(* Logix 5000 project; controller ToyPlant Emulate 5570 rev 30.12; software revision 30.00 *)

TASK MainTask (continuous, watchdog 500 ms) : MainProgram

MODULES
   Local : Emulate 5570 (ICP 2, rev 30.12)
END_MODULES

PROGRAM MainProgram   (* main routine MainRoutine *)
VAR
   Action_000 : SFC_ACTION := (Count := 2);
   Action_001 : SFC_ACTION := (Count := 1);
   Action_002 : SFC_ACTION := (Count := 1);
   Action_003 : SFC_ACTION := (Count := 1);
   Action_004 : SFC_ACTION := (Count := 1);
   Action_005 : SFC_ACTION := (Count := 14);
   Action_006 : SFC_ACTION := (Count := 1);
   Action_007 : SFC_ACTION := (Count := 1);
   Action_008 : SFC_ACTION := (Count := 1);
   Action_009 : SFC_ACTION := (Count := 1);
   Action_010 : SFC_ACTION := (Count := 1);
   Action_011 : SFC_ACTION := (Count := 2);
   Action_012 : SFC_ACTION := (Count := 2);
   Action_013 : SFC_ACTION := (Count := 1);
   Action_014 : SFC_ACTION := (Count := 1);
   Action_015 : SFC_ACTION := (Count := 1);
   Action_016 : SFC_ACTION := (Count := 1);
   Action_017 : SFC_ACTION := (Count := 1);
   Action_018 : SFC_ACTION := (Count := 1);
   Action_019 : SFC_ACTION := (Count := 1);
   Action_020 : SFC_ACTION := (Count := 1);
   Action_021 : SFC_ACTION := (Status := 16#0020_0000, PauseTimer := 1, Count := 1);
   Action_022 : SFC_ACTION;
   Action_023 : SFC_ACTION;
   Action_024 : SFC_ACTION;
   Action_025 : SFC_ACTION;
   Action_026 : SFC_ACTION;
   Action_027 : SFC_ACTION;
   Action_028 : SFC_ACTION;
   Action_029 : SFC_ACTION := (Status := 16#0020_0000, PauseTimer := 1);
   Action_030 : SFC_ACTION := (Status := 16#0020_0000, PauseTimer := 1);
   Action_031 : SFC_ACTION := (Status := 16#0020_0000, PauseTimer := 1);
   Action_032 : SFC_ACTION := (Status := 16#0020_0000, PauseTimer := 1);
   Action_033 : SFC_ACTION := (Status := 16#0020_0000, PauseTimer := 1);
   Action_034 : SFC_ACTION := (Status := 16#0020_0000, PauseTimer := 1);
   Action_035 : SFC_ACTION := (Status := 16#0020_0000, PauseTimer := 1);
   Action_036 : SFC_ACTION := (Status := 16#0020_0000, PauseTimer := 1);
   Action_037 : SFC_ACTION := (Status := 16#0020_0000, PauseTimer := 1);
   Action_038 : SFC_ACTION := (Status := 16#0020_0000, PauseTimer := 1);
   Action_039 : SFC_ACTION := (Status := 16#0020_0000, PauseTimer := 1);
   Action_040 : SFC_ACTION := (Status := 16#0020_0000, PauseTimer := 1);
   Action_041 : SFC_ACTION := (Status := 16#0020_0000, PauseTimer := 1);
   Action_042 : SFC_ACTION := (Status := 16#0020_0000, PauseTimer := 1);
   Action_043 : SFC_ACTION := (Status := 16#0020_0000, PauseTimer := 1);
   Action_044 : SFC_ACTION := (Status := 16#0020_0000, PauseTimer := 1);
   Action_045 : SFC_ACTION := (Status := 16#0020_0000, PauseTimer := 1);
   BarcoReady : BOOL;
   CasaReady : BOOL;
   ContadorBarco : COUNTER := (PRE := 25);
   ContadorCasa : COUNTER := (PRE := 25);
   ContadorJuguetes : COUNTER := (PRE := 4);
   ContadorMoldes : COUNTER := (PRE := 4);
   ContadorMoto : COUNTER := (PRE := 25);
   MotoReady : BOOL;
   Off_ServoWorking : BOOL;
   PresetBarco : DINT := 1000;
   PresetCasa : DINT := 1000;
   PresetMoto : DINT := 1000;
   Step_000 : SFC_STEP := (T := 14169, TMax := 14169, Count := 2);
   Step_001 : SFC_STEP := (T := 1304, TMax := 1304, Count := 1);
   Step_002 : SFC_STEP := (T := 2486, TMax := 2486, Count := 1);
   Step_003 : SFC_STEP := (T := 21, TMax := 21, Count := 1);
   Step_004 : SFC_STEP := (T := 1039, TMax := 1039, Count := 1);
   Step_005 : SFC_STEP := (T := 21, TMax := 22, Count := 14);
   Step_006 : SFC_STEP := (T := 1975, TMax := 1975, Count := 1);
   Step_007 : SFC_STEP := (T := 1331, TMax := 1331, Count := 1);
   Step_008 : SFC_STEP := (T := 1030, TMax := 1030, Count := 1);
   Step_009 : SFC_STEP := (T := 1031, TMax := 1031, Count := 1);
   Step_010 : SFC_STEP := (T := 50, TMax := 50, Count := 1);
   Step_011 : SFC_STEP := (T := 1037, TMax := 1037, Count := 2);
   Step_012 : SFC_STEP := (T := 15933, TMax := 15933, Count := 2);
   Step_013 : SFC_STEP := (T := 1034, TMax := 1034, Count := 1);
   Step_014 : SFC_STEP := (T := 1032, TMax := 1032, Count := 1);
   Step_015 : SFC_STEP := (T := 1034, TMax := 1034, Count := 1);
   Step_016 : SFC_STEP := (T := 22, TMax := 22, Count := 1);
   Step_017 : SFC_STEP := (T := 1034, TMax := 1034, Count := 1);
   Step_018 : SFC_STEP := (T := 1031, TMax := 1031, Count := 1);
   Step_019 : SFC_STEP := (T := 1031, TMax := 1031, Count := 1);
   Step_020 : SFC_STEP := (T := 50, TMax := 50, Count := 1);
   Step_021 : SFC_STEP := (Status := 16#0820_0201, DN := 1, PauseTimer := 1, T := 21, TMax := 21, Count := 1);
   Step_022 : SFC_STEP;
   Step_023 : SFC_STEP;
   Step_024 : SFC_STEP;
   Step_025 : SFC_STEP;
   Step_026 : SFC_STEP;
   Step_027 : SFC_STEP;
   Step_028 : SFC_STEP;
   Step_029 : SFC_STEP := (Status := 16#0020_0000, PauseTimer := 1);
   Step_030 : SFC_STEP := (Status := 16#0020_0000, PauseTimer := 1);
   Step_031 : SFC_STEP := (Status := 16#0020_0000, PauseTimer := 1);
   Step_032 : SFC_STEP := (Status := 16#0020_0000, PauseTimer := 1);
   Step_033 : SFC_STEP := (Status := 16#0020_0000, PauseTimer := 1);
   Step_034 : SFC_STEP := (Status := 16#0020_0000, PauseTimer := 1);
   Step_035 : SFC_STEP := (Status := 16#0020_0000, PauseTimer := 1);
   Step_036 : SFC_STEP := (Status := 16#0020_0000, PauseTimer := 1);
   Step_037 : SFC_STEP := (Status := 16#0020_0000, PauseTimer := 1);
   Step_038 : SFC_STEP := (Status := 16#0020_0000, PauseTimer := 1);
   Step_039 : SFC_STEP := (Status := 16#0020_0000, PauseTimer := 1);
   Step_040 : SFC_STEP := (Status := 16#0020_0000, PauseTimer := 1);
   Step_041 : SFC_STEP := (Status := 16#0020_0000, PauseTimer := 1);
   Step_042 : SFC_STEP := (Status := 16#0020_0000, PauseTimer := 1);
   Step_043 : SFC_STEP := (Status := 16#0020_0000, PauseTimer := 1);
   Step_044 : SFC_STEP := (Status := 16#0020_0000, PauseTimer := 1);
   Step_045 : SFC_STEP := (Status := 16#0020_0000, PauseTimer := 1);
   Step_046 : SFC_STEP := (Status := 16#0020_0000, PauseTimer := 1);
   Stop_000 : SFC_STOP := (Status := 16#a000_2001, X := 1);
   Stop_001 : SFC_STOP;
   TimerBarco_1 : FBD_TIMER := (TimerEnable := 1, PRE := 1000, ACC := 1015, EN := 1, DN := 1);
   TimerBarco_2 : FBD_TIMER := (TimerEnable := 1, PRE := 1000, Reset := 1, ACC := 1013, EN := 1, DN := 1);
   TimerBarco_3 : FBD_TIMER := (TimerEnable := 1, PRE := 1000, ACC := 1011, EN := 1, DN := 1);
   TimerBarco_4 : FBD_TIMER := (TimerEnable := 1, PRE := 1000, ACC := 1014, EN := 1, DN := 1);
   TimerBarco_5 : FBD_TIMER := (TimerEnable := 1, PRE := 1000, ACC := 1013, EN := 1, DN := 1);
   TimerBarco_6 : FBD_TIMER := (TimerEnable := 1, PRE := 1000, ACC := 1000, EN := 1, DN := 1);
   TimerBarco_7 : FBD_TIMER := (TimerEnable := 1, PRE := 1000, ACC := 1010, EN := 1, DN := 1);
   TimerCasa_1 : FBD_TIMER := (TimerEnable := 1, PRE := 1000, ACC := 1015, EN := 1, DN := 1);
   TimerCasa_2 : FBD_TIMER := (TimerEnable := 1, PRE := 1000, ACC := 1015, EN := 1, DN := 1);
   TimerCasa_3 : FBD_TIMER := (TimerEnable := 1, PRE := 1000, ACC := 1015, EN := 1, DN := 1);
   TimerCasa_4 : FBD_TIMER := (TimerEnable := 1, PRE := 1000, ACC := 1015, EN := 1, DN := 1);
   TimerCasa_5 : FBD_TIMER := (TimerEnable := 1, PRE := 1000, ACC := 1015, EN := 1, DN := 1);
   TimerDespacho_1 : FBD_TIMER;
   TimerDespacho_2 : FBD_TIMER;
   TimerDespacho_3 : FBD_TIMER;
   TimerDespacho_4 : FBD_TIMER;
   TimerDespacho_5 : FBD_TIMER;
   TimerMoto_1 : FBD_TIMER := (TimerEnable := 1, PRE := 1000, ACC := 1015, EN := 1, DN := 1);
   TimerMoto_2 : FBD_TIMER := (TimerEnable := 1, PRE := 1000, ACC := 1018, EN := 1, DN := 1);
   TimerMoto_3 : FBD_TIMER := (TimerEnable := 1, PRE := 1300, ACC := 1310, EN := 1, DN := 1);
   TimerMoto_4 : FBD_TIMER := (TimerEnable := 1, PRE := 1000, ACC := 1000, EN := 1, DN := 1);
   TimerMoto_5 : FBD_TIMER := (TimerEnable := 1, PRE := 1000, ACC := 1010, EN := 1, DN := 1);
   TimerMoto_6 : FBD_TIMER := (TimerEnable := 1, PRE := 1000, ACC := 1013, EN := 1, DN := 1);
   TimerMoto_7 : FBD_TIMER;
   TimerPickBarco : TIMER := (PRE := 1000);
   TimerPickcasa : TIMER := (PRE := 1000);
   TimerPickMoto : TIMER := (PRE := 1000);
   Tran_000 : BOOL;
   Tran_001 : BOOL := 1;
   Tran_002 : BOOL := 1;
   Tran_003 : BOOL := 1;
   Tran_004 : BOOL := 1;
   Tran_005 : BOOL := 1;
   Tran_006 : BOOL := 1;
   Tran_007 : BOOL := 1;
   Tran_008 : BOOL := 1;
   Tran_009 : BOOL := 1;
   Tran_010 : BOOL := 1;
   Tran_011 : BOOL := 1;
   Tran_012 : BOOL;
   Tran_013 : BOOL := 1;
   Tran_014 : BOOL := 1;
   Tran_015 : BOOL := 1;
   Tran_016 : BOOL := 1;
   Tran_017 : BOOL := 1;
   Tran_018 : BOOL := 1;
   Tran_019 : BOOL := 1;
   Tran_020 : BOOL := 1;
   Tran_021 : BOOL := 1;
   Tran_022 : BOOL;
   Tran_023 : BOOL;
   Tran_024 : BOOL;
   Tran_025 : BOOL;
   Tran_026 : BOOL;
   Tran_027 : BOOL;
   Tran_028 : BOOL;
   Tran_029 : BOOL;
   Tran_030 : BOOL;
   Tran_031 : BOOL;
   Tran_032 : BOOL;
   Tran_033 : BOOL;
   Tran_034 : BOOL;
   Tran_035 : BOOL;
   Tran_036 : BOOL;
   Tran_037 : BOOL;
   Tran_038 : BOOL;
   Tran_039 : BOOL;
   Tran_040 : BOOL;
   Tran_041 : BOOL;
   Tran_042 : BOOL;
   Tran_043 : BOOL;
   Tran_044 : BOOL;
   Tran_045 : BOOL;
   Tran_046 : BOOL;
   Tran_047 : BOOL;
   Tran_048 : BOOL;
   Tran_049 : BOOL;
END_VAR
VAR_OUTPUT
   Ajuste_Cero : BOOL; {access Read Only}
   Ajuste_Pos1 : BOOL; {access Read Only}
   AjusteCasa_Cero : BOOL; {access Read Only}
   AjusteCasa_Pos1 : BOOL; {access Read Only}
   BarcoACaja : BOOL := 1; {access Read Only}
   BarcosAPick : BOOL; {access Read Only}
   CalidadYEmpaquetado : BOOL; {access Read Only}
   CasaACaja : BOOL := 1; {access Read Only}
   CasasAPick : BOOL; {access Read Only}
   Chasis_Cero : BOOL := 1; {access Read Only}
   Chasis_Pos1 : BOOL; {access Read Only}
   Dispensar_CajaBarcos : BOOL;
   Dispensar_CajaCasas : BOOL;
   Dispensar_CajaMotos : BOOL;
   Dispensar_Chasis : BOOL; {access Read Only}
   Dispensar_Inf : BOOL; {access Read Only}
   Dispensar_Paredes : BOOL; {access Read Only}
   Dispensar_Ruedas : BOOL; {access Read Only}
   Dispensar_Sup : BOOL; {access Read Only}
   Dispensar_Techo : BOOL; {access Read Only}
   Dispensar_Timon : BOOL; {access Read Only}
   EnsamblePrevio : BOOL; {access Read Only}
   EnsambleYPintado : BOOL; {access Read Only}
   Inf_Cero : BOOL; {access Read Only}
   Inf_Pos1 : BOOL; {access Read Only}
   Listas : BOOL; {access Read Only}
   MotoACaja : BOOL := 1; {access Read Only}
   MotosAPick : BOOL; {access Read Only}
   Paredes_Cero : BOOL; {access Read Only}
   Paredes_Pos1 : BOOL; {access Read Only}
   PiezasAzules : BOOL; {access Read Only}
   PiezasNegras : BOOL; {access Read Only}
   PiezasRojas : BOOL; {access Read Only}
   PuertaBarco : BOOL; {access Read Only}
   PuertaCasa : BOOL; {access Read Only}
   PuertaMoto : BOOL; {access Read Only}
   RUNNING : BOOL; {access Read Only}
   SeparadoYAcabado : BOOL; {access Read Only}
   Servo_PosBarco : BOOL; {access Read Only}
   Servo_PosCasa : BOOL; {access Read Only}
   Servo_PosMoto : BOOL; {access Read Only}
   Sup_Cero : BOOL; {access Read Only}
   Sup_Pos1 : BOOL; {access Read Only}
   Techo_Cero : BOOL; {access Read Only}
   Techo_Pos1 : BOOL; {access Read Only}
   Timon_Cero : BOOL; {access Read Only}
   Timon_Pos1 : BOOL; {access Read Only}
END_VAR
VAR_INPUT
   Chasis_Ubicado : BOOL;
   EntradaMolde : BOOL;
   Inf_Ubicado : BOOL;
   JugueteEnPosicion : BOOL;
   OnCalEmp : BOOL;
   OnEnsamPin : BOOL;
   OnListas : BOOL;
   OnPre : BOOL;
   OnSepAca : BOOL;
   Paredes_Ubicadas : BOOL;
   Ruedas1_Ubicadas : BOOL;
   Ruedas2_Ubicadas : BOOL;
   Ruedas_Cero : BOOL := 1;
   Ruedas_Pos1 : BOOL;
   Ruedas_Pos2 : BOOL;
   SaleBarco : BOOL;
   SaleCasa : BOOL;
   SaleMoto : BOOL;
   START_PROCESS : BOOL;
   STOP_ALL : BOOL := 1;
   Sup_Ubicado : BOOL;
   Techo_Ubicado : BOOL;
   Timon_Ubicado : BOOL;
END_VAR

ROUTINE Bandas   (* ladder *)
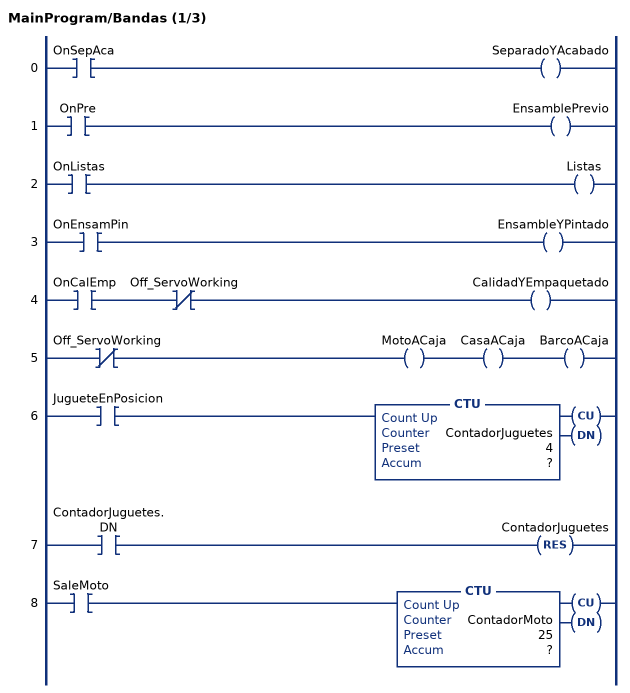
   0: XIC(OnSepAca)OTE(SeparadoYAcabado);
   1: XIC(OnPre)OTE(EnsamblePrevio);
   2: XIC(OnListas)OTE(Listas);
   3: XIC(OnEnsamPin)OTE(EnsambleYPintado);
   4: XIC(OnCalEmp)XIO(Off_ServoWorking)OTE(CalidadYEmpaquetado);
   5: XIO(Off_ServoWorking)OTE(MotoACaja)OTE(CasaACaja)OTE(BarcoACaja);
   6: XIC(JugueteEnPosicion)CTU(ContadorJuguetes,?,?);
   7: XIC(ContadorJuguetes.DN)RES(ContadorJuguetes);
   8: XIC(SaleMoto)CTU(ContadorMoto,?,?);
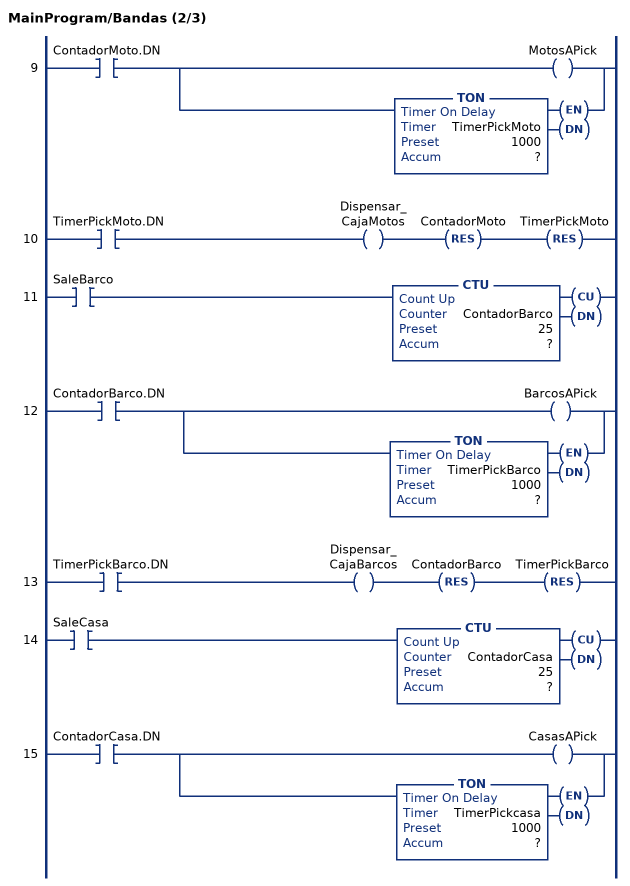
   9: XIC(ContadorMoto.DN)[OTE(MotosAPick) ,TON(TimerPickMoto,?,?) ];
   10: XIC(TimerPickMoto.DN)OTE(Dispensar_CajaMotos)RES(ContadorMoto)RES(TimerPickMoto);
   11: XIC(SaleBarco)CTU(ContadorBarco,?,?);
   12: XIC(ContadorBarco.DN)[OTE(BarcosAPick) ,TON(TimerPickBarco,?,?) ];
   13: XIC(TimerPickBarco.DN)OTE(Dispensar_CajaBarcos)RES(ContadorBarco)RES(TimerPickBarco);
   14: XIC(SaleCasa)CTU(ContadorCasa,?,?);
   15: XIC(ContadorCasa.DN)[OTE(CasasAPick) ,TON(TimerPickcasa,?,?) ];
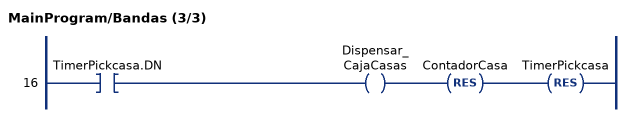
   16: XIC(TimerPickcasa.DN)OTE(Dispensar_CajaCasas)RES(ContadorCasa)RES(TimerPickcasa);
END_ROUTINE

ROUTINE Despacho   (* sequential function chart *)
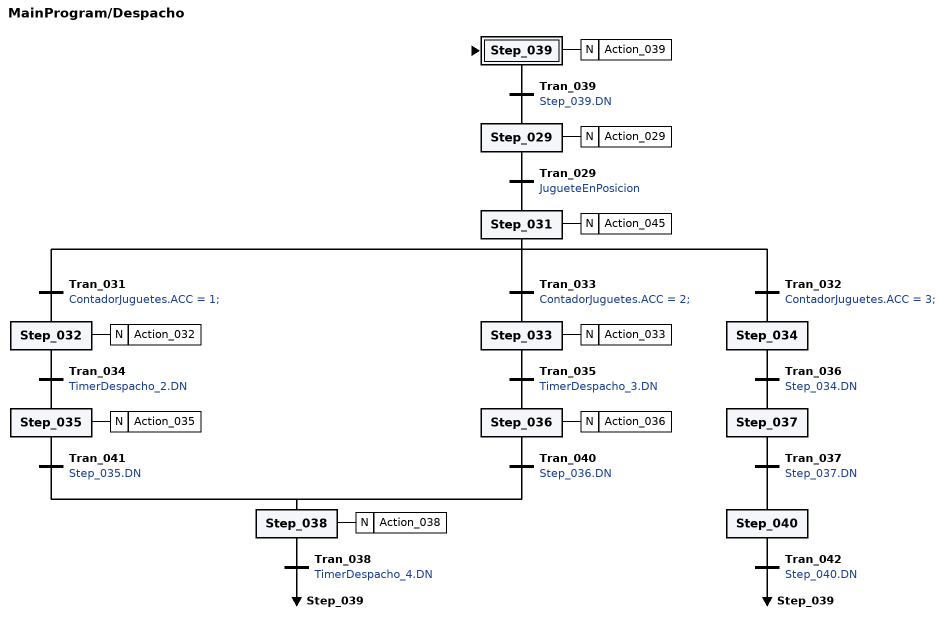
   INITIAL_STEP Step_039:
      ACTION Action_039 (N):
         TimerDespacho_1.Reset := 1;
         TimerDespacho_2.Reset := 1;
         TimerDespacho_3.Reset := 1;
         TimerDespacho_4.Reset := 1;
         TimerDespacho_5.Reset := 1;
      END_ACTION
   END_STEP
   TRANSITION Tran_039 FROM Step_039 TO Step_029
      := Step_039.DN
   END_TRANSITION
   STEP Step_029:
      ACTION Action_029 (N):
         Off_ServoWorking := 0;
         Servo_PosMoto := 0;
      END_ACTION
   END_STEP
   TRANSITION Tran_029 FROM Step_029 TO Step_031
      := JugueteEnPosicion
   END_TRANSITION
   STEP Step_031:
      ACTION Action_045 (N):
         Off_ServoWorking := 1;
      END_ACTION
   END_STEP
   TRANSITION Tran_031 FROM Step_031 TO Step_032
      := ContadorJuguetes.ACC = 1;
   END_TRANSITION
   TRANSITION Tran_033 FROM Step_031 TO Step_033
      := ContadorJuguetes.ACC = 2;
   END_TRANSITION
   TRANSITION Tran_032 FROM Step_031 TO Step_034
      := ContadorJuguetes.ACC = 3;
   END_TRANSITION
   STEP Step_032:
      ACTION Action_032 (N):
         Servo_PosCasa := 1;
         
         TimerDespacho_2.Reset := 0;
         TimerDespacho_2.TimerEnable := 1;
         TONR(TimerDespacho_2);
         TimerDespacho_2.PRE := 1000;
      END_ACTION
   END_STEP
   STEP Step_033:
      ACTION Action_033 (N):
         Servo_PosBarco := 1;
         
         
         TimerDespacho_3.Reset := 0;
         TimerDespacho_3.TimerEnable := 1;
         TONR(TimerDespacho_3);
         TimerDespacho_3.PRE := 1000;
      END_ACTION
   END_STEP
   STEP Step_034:
   END_STEP
   TRANSITION Tran_034 FROM Step_032 TO Step_035
      := TimerDespacho_2.DN
   END_TRANSITION
   TRANSITION Tran_035 FROM Step_033 TO Step_036
      := TimerDespacho_3.DN
   END_TRANSITION
   TRANSITION Tran_036 FROM Step_034 TO Step_037
      := Step_034.DN
   END_TRANSITION
   STEP Step_035:
      ACTION Action_035 (N):
         Servo_PosCasa := 0;
      END_ACTION
   END_STEP
   STEP Step_036:
      ACTION Action_036 (N):
         Servo_PosBarco := 0;
      END_ACTION
   END_STEP
   STEP Step_037:
   END_STEP
   TRANSITION Tran_041 FROM Step_035 TO Step_038
      := Step_035.DN
   END_TRANSITION
   TRANSITION Tran_040 FROM Step_036 TO Step_038
      := Step_036.DN
   END_TRANSITION
   TRANSITION Tran_037 FROM Step_037 TO Step_040
      := Step_037.DN
   END_TRANSITION
   STEP Step_038:
      ACTION Action_038 (N):
         Servo_PosMoto := 1;
         
         TimerDespacho_4.Reset := 0;
         TimerDespacho_4.TimerEnable := 1;
         TONR(TimerDespacho_4);
         TimerDespacho_4.PRE := 1000;
      END_ACTION
   END_STEP
   STEP Step_040:
   END_STEP
   TRANSITION Tran_038 FROM Step_038 TO Step_039
      := TimerDespacho_4.DN
   END_TRANSITION
   TRANSITION Tran_042 FROM Step_040 TO Step_039
      := Step_040.DN
   END_TRANSITION
END_ROUTINE

ROUTINE EnsambleBarco   (* sequential function chart *)
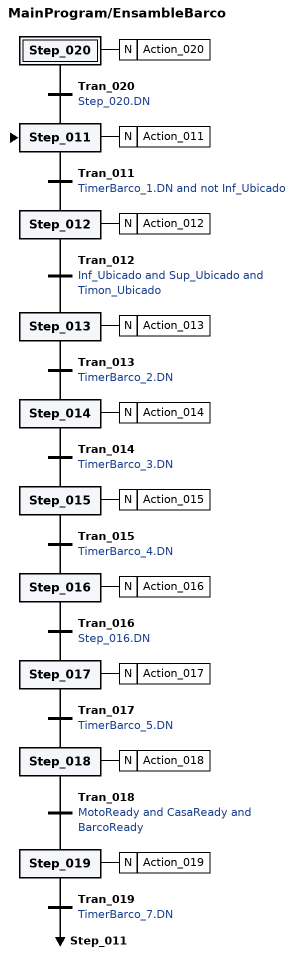
   INITIAL_STEP Step_020:
      ACTION Action_020 (N):
         TimerBarco_1.Reset := 1;
         TimerBarco_2.Reset := 1;
         TimerBarco_3.Reset := 1;
         TimerBarco_4.Reset := 1;
         TimerBarco_5.Reset := 1;
         TimerBarco_6.Reset := 1;
         TimerBarco_7.Reset := 1;
      END_ACTION
   END_STEP
   TRANSITION Tran_020 FROM Step_020 TO Step_011
      := Step_020.DN
   END_TRANSITION
   STEP Step_011:
      ACTION Action_011 (N):
         Inf_Cero := 1; Sup_Cero := 1; Timon_Cero := 1; Ajuste_Cero := 1; PuertaBarco := 1;
         Dispensar_Inf := 0; Dispensar_Sup := 0; Dispensar_Timon := 0;
         
         TimerBarco_1.Reset := 0;
         TimerBarco_1.TimerEnable := 1;
         TONR(TimerBarco_1);
         TimerBarco_1.PRE := PresetBarco;
         
         TimerBarco_2.Reset := 1;
      END_ACTION
   END_STEP
   TRANSITION Tran_011 FROM Step_011 TO Step_012
      := TimerBarco_1.DN and not Inf_Ubicado
         
   END_TRANSITION
   STEP Step_012:
      ACTION Action_012 (N):
         Dispensar_Inf := 1; Dispensar_Sup := 1; Dispensar_Timon := 1;
         Inf_Cero := 0; Sup_Cero := 0; Timon_Cero := 0; Ajuste_Cero := 0;
      END_ACTION
   END_STEP
   TRANSITION Tran_012 FROM Step_012 TO Step_013
      := Inf_Ubicado and Sup_Ubicado and Timon_Ubicado
   END_TRANSITION
   STEP Step_013:
      ACTION Action_013 (N):
         Dispensar_Inf := 0; Dispensar_Sup := 0; Dispensar_Timon := 0;
         Inf_Pos1 := 1;
         
         TimerBarco_2.Reset := 0;
         TimerBarco_2.TimerEnable := 1;
         TONR(TimerBarco_2);
         TimerBarco_2.PRE := PresetBarco;
         
         TimerBarco_3.Reset := 1;
      END_ACTION
   END_STEP
   TRANSITION Tran_013 FROM Step_013 TO Step_014
      := TimerBarco_2.DN
   END_TRANSITION
   STEP Step_014:
      ACTION Action_014 (N):
         Inf_Pos1 := 0; Sup_Pos1 := 1;
         
         TimerBarco_3.Reset := 0;
         TimerBarco_3.TimerEnable := 1;
         TONR(TimerBarco_3);
         TimerBarco_3.PRE := PresetBarco;
         
         TimerBarco_4.Reset := 1;
      END_ACTION
   END_STEP
   TRANSITION Tran_014 FROM Step_014 TO Step_015
      := TimerBarco_3.DN
   END_TRANSITION
   STEP Step_015:
      ACTION Action_015 (N):
         Sup_Pos1 := 0; Timon_Pos1 := 1;
         
         TimerBarco_4.Reset := 0;
         TimerBarco_4.TimerEnable := 1;
         TONR(TimerBarco_4);
         TimerBarco_4.PRE := PresetBarco;
         
         TimerBarco_5.Reset := 1;
      END_ACTION
   END_STEP
   TRANSITION Tran_015 FROM Step_015 TO Step_016
      := TimerBarco_4.DN
   END_TRANSITION
   STEP Step_016:
      ACTION Action_016 (N):
         Timon_Pos1 := 0;
      END_ACTION
   END_STEP
   TRANSITION Tran_016 FROM Step_016 TO Step_017
      := Step_016.DN
   END_TRANSITION
   STEP Step_017:
      ACTION Action_017 (N):
         Timon_Cero := 1;
         
         TimerBarco_5.Reset := 0;
         TimerBarco_5.TimerEnable := 1;
         TONR(TimerBarco_5);
         TimerBarco_5.PRE := PresetBarco;
         
         TimerBarco_6.Reset := 1;
      END_ACTION
   END_STEP
   TRANSITION Tran_017 FROM Step_017 TO Step_018
      := TimerBarco_5.DN
   END_TRANSITION
   STEP Step_018:
      ACTION Action_018 (N):
         Timon_Cero := 0; Ajuste_Pos1 := 1;
         
         BarcoReady := 1;
         
         TimerBarco_7.Reset := 1;
      END_ACTION
   END_STEP
   TRANSITION Tran_018 FROM Step_018 TO Step_019
      := MotoReady and CasaReady and BarcoReady
   END_TRANSITION
   STEP Step_019:
      ACTION Action_019 (N):
         Ajuste_Pos1 := 0;
         PuertaBarco :=0;
         BarcoReady := 0;
         
         TimerBarco_7.Reset := 0;
         TimerBarco_7.TimerEnable := 1;
         TONR(TimerBarco_7);
         TimerBarco_7.PRE := PresetBarco;
         
         TimerBarco_1.Reset := 1;
      END_ACTION
   END_STEP
   TRANSITION Tran_019 FROM Step_019 TO Step_011
      := TimerBarco_7.DN
   END_TRANSITION
END_ROUTINE

ROUTINE EnsambleCasa   (* sequential function chart *)
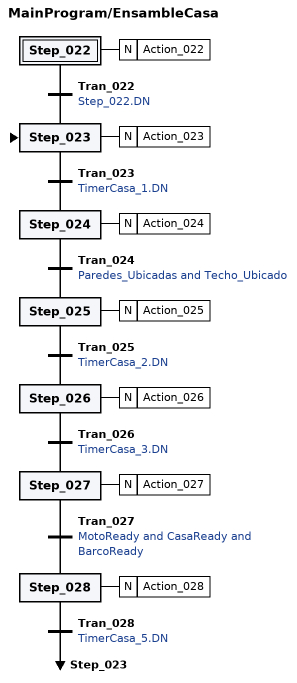
   INITIAL_STEP Step_022:
      ACTION Action_022 (N):
         TimerCasa_1.Reset := 1; TimerCasa_2.Reset := 1; TimerCasa_3.Reset := 1; TimerCasa_4.Reset := 1;
         TimerCasa_5.Reset := 1;
      END_ACTION
   END_STEP
   TRANSITION Tran_022 FROM Step_022 TO Step_023
      := Step_022.DN
   END_TRANSITION
   STEP Step_023:
      ACTION Action_023 (N):
         Paredes_Cero := 1; Techo_Cero := 1; AjusteCasa_Cero := 1; PuertaCasa := 1;
         
         TimerCasa_1.Reset := 0;
         TimerCasa_1.TimerEnable := 1;
         TONR(TimerCasa_1);
         TimerCasa_1.PRE := PresetCasa;
         
         TimerCasa_2.Reset := 1;
      END_ACTION
   END_STEP
   TRANSITION Tran_023 FROM Step_023 TO Step_024
      := TimerCasa_1.DN
   END_TRANSITION
   STEP Step_024:
      ACTION Action_024 (N):
         Paredes_Cero := 0; Techo_Cero := 0; AjusteCasa_Cero := 0; Dispensar_Paredes := 1; Dispensar_Techo := 1;
      END_ACTION
   END_STEP
   TRANSITION Tran_024 FROM Step_024 TO Step_025
      := Paredes_Ubicadas and Techo_Ubicado
   END_TRANSITION
   STEP Step_025:
      ACTION Action_025 (N):
         Dispensar_Paredes := 0; Dispensar_Techo := 0; Paredes_Pos1 := 1;
         
         TimerCasa_2.Reset := 0;
         TimerCasa_2.TimerEnable := 1;
         TONR(TimerCasa_2);
         TimerCasa_2.PRE := PresetCasa;
         
         TimerCasa_3.Reset := 1;
      END_ACTION
   END_STEP
   TRANSITION Tran_025 FROM Step_025 TO Step_026
      := TimerCasa_2.DN
   END_TRANSITION
   STEP Step_026:
      ACTION Action_026 (N):
         Paredes_Pos1 := 0; Techo_Pos1 := 1;
         
         TimerCasa_3.Reset := 0;
         TimerCasa_3.TimerEnable := 1;
         TONR(TimerCasa_3);
         TimerCasa_3.PRE := PresetCasa;
         
         TimerCasa_4.Reset := 1;
      END_ACTION
   END_STEP
   TRANSITION Tran_026 FROM Step_026 TO Step_027
      := TimerCasa_3.DN
   END_TRANSITION
   STEP Step_027:
      ACTION Action_027 (N):
         AjusteCasa_Pos1 := 1;
         Techo_Pos1 := 0;
         
         CasaReady := 1;
         
         TimerCasa_5.Reset := 1;
      END_ACTION
   END_STEP
   TRANSITION Tran_027 FROM Step_027 TO Step_028
      := MotoReady and CasaReady and BarcoReady
   END_TRANSITION
   STEP Step_028:
      ACTION Action_028 (N):
         AjusteCasa_Pos1 := 0;
         PuertaCasa := 0;
         CasaReady := 0;
         
         TimerCasa_5.Reset := 0;
         TimerCasa_5.TimerEnable := 1;
         TONR(TimerCasa_5);
         TimerCasa_5.PRE := PresetCasa;
         
         TimerCasa_1.Reset := 1;
      END_ACTION
   END_STEP
   TRANSITION Tran_028 FROM Step_028 TO Step_023
      := TimerCasa_5.DN
   END_TRANSITION
END_ROUTINE

ROUTINE EnsambleMoto   (* sequential function chart *)
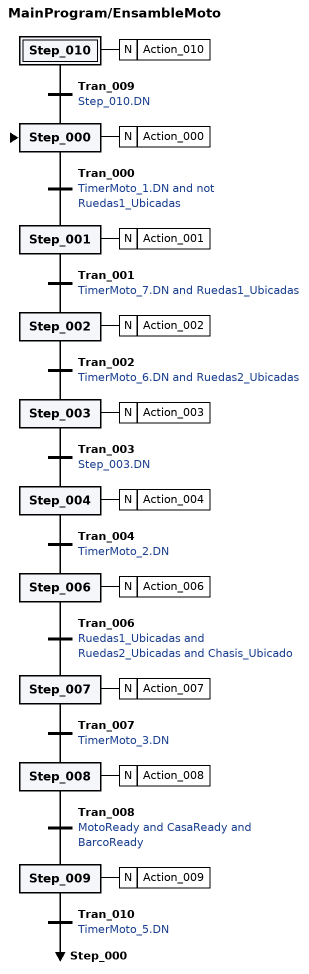
   INITIAL_STEP Step_010:
      ACTION Action_010 (N):
         TimerMoto_1.Reset := 1;
         TimerMoto_2.Reset := 1;
         TimerMoto_3.Reset := 1;
         TimerMoto_4.Reset := 1;
         TimerMoto_5.Reset := 1;
         TimerMoto_6.Reset := 1;
      END_ACTION
   END_STEP
   TRANSITION Tran_009 FROM Step_010 TO Step_000
      := Step_010.DN
         
   END_TRANSITION
   STEP Step_000:
      ACTION Action_000 (N):
         Chasis_Cero := 1;
         Ruedas_Cero := 1;
         PuertaMoto := 1;
         Dispensar_Ruedas := 0;
         Dispensar_Chasis := 0;
         
         TimerMoto_1.Reset := 0;
         TimerMoto_1.TimerEnable := 1;
         TONR(TimerMoto_1);
         TimerMoto_1.PRE := PresetMoto;
         
         TimerMoto_7.Reset := 1;
      END_ACTION
   END_STEP
   TRANSITION Tran_000 FROM Step_000 TO Step_001
      := TimerMoto_1.DN and not Ruedas1_Ubicadas
   END_TRANSITION
   STEP Step_001:
      ACTION Action_001 (N):
         Dispensar_Ruedas := 1;
         Dispensar_Chasis := 1;
         Chasis_Cero := 0;
         Ruedas_Cero := 0;
         
         TimerMoto_6.Reset := 1;
         
         TimerMoto_7.Reset := 0;
         TimerMoto_7.TimerEnable := 1;
         TONR(TimerMoto_7);
         TimerMoto_7.PRE := PresetMoto;
      END_ACTION
   END_STEP
   TRANSITION Tran_001 FROM Step_001 TO Step_002
      := TimerMoto_7.DN and Ruedas1_Ubicadas
         
   END_TRANSITION
   STEP Step_002:
      ACTION Action_002 (N):
         Ruedas_Pos2 := 1;
         Dispensar_Ruedas := 0;
         Dispensar_Chasis := 0;
         
         TimerMoto_6.Reset := 0;
         TimerMoto_6.TimerEnable := 1;
         TONR(TimerMoto_6);
         TimerMoto_6.PRE := PresetMoto;
      END_ACTION
   END_STEP
   TRANSITION Tran_002 FROM Step_002 TO Step_003
      := TimerMoto_6.DN and Ruedas2_Ubicadas
   END_TRANSITION
   STEP Step_003:
      ACTION Action_003 (N):
         Ruedas_Pos2 := 0;
         TimerMoto_2.Reset := 1;
      END_ACTION
   END_STEP
   TRANSITION Tran_003 FROM Step_003 TO Step_004
      := Step_003.DN
   END_TRANSITION
   STEP Step_004:
      ACTION Action_004 (N):
         Ruedas_Cero := 1;
         
         TimerMoto_2.Reset := 0;
         TimerMoto_2.TimerEnable := 1;
         TONR(TimerMoto_2);
         TimerMoto_2.PRE := PresetMoto;
      END_ACTION
   END_STEP
   TRANSITION Tran_004 FROM Step_004 TO Step_006
      := TimerMoto_2.DN
   END_TRANSITION
   STEP Step_006:
      ACTION Action_006 (N):
         Ruedas_Cero := 0; Dispensar_Ruedas := 1; TimerMoto_3.Reset := 1;
      END_ACTION
   END_STEP
   TRANSITION Tran_006 FROM Step_006 TO Step_007
      := Ruedas1_Ubicadas and Ruedas2_Ubicadas and Chasis_Ubicado
   END_TRANSITION
   STEP Step_007:
      ACTION Action_007 (N):
         Chasis_Pos1 := 1;
         Dispensar_Ruedas := 0;
         
         TimerMoto_3.Reset := 0;
         TimerMoto_3.TimerEnable := 1;
         TONR(TimerMoto_3);
         TimerMoto_3.PRE := PresetMoto;
         
         TimerMoto_4.Reset := 1;
      END_ACTION
   END_STEP
   TRANSITION Tran_007 FROM Step_007 TO Step_008
      := TimerMoto_3.DN
   END_TRANSITION
   STEP Step_008:
      ACTION Action_008 (N):
         Ruedas_Pos1 := 1;
         Chasis_Pos1 := 0;
         
         MotoReady := 1;
         
         TimerMoto_5.Reset := 1;
      END_ACTION
   END_STEP
   TRANSITION Tran_008 FROM Step_008 TO Step_009
      := MotoReady and CasaReady and BarcoReady
         
   END_TRANSITION
   STEP Step_009:
      ACTION Action_009 (N):
         Ruedas_Pos1 := 0;
         PuertaMoto := 0;
         MotoReady := 0;
         
         TimerMoto_5.Reset := 0;
         TimerMoto_5.TimerEnable := 1;
         TONR(TimerMoto_5);
         TimerMoto_5.PRE := PresetMoto;
         
         TimerMoto_1.Reset := 1;
      END_ACTION
   END_STEP
   TRANSITION Tran_010 FROM Step_009 TO Step_000
      := TimerMoto_5.DN
         
   END_TRANSITION
END_ROUTINE

ROUTINE MainRoutine   (* ladder *)
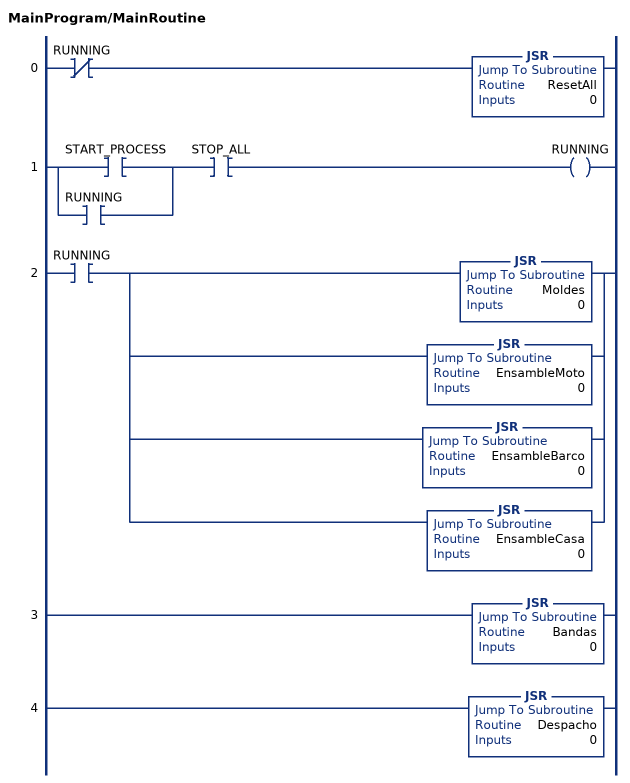
   0: XIO(RUNNING)JSR(ResetAll,0);
   1: [XIC(START_PROCESS) ,XIC(RUNNING) ]XIC(STOP_ALL)OTE(RUNNING);
   2: XIC(RUNNING)[JSR(Moldes,0) ,[JSR(EnsambleMoto,0) ,[JSR(EnsambleBarco,0) ,JSR(EnsambleCasa,0) ] ] ];
   3: JSR(Bandas,0);
   4: JSR(Despacho,0);
END_ROUTINE

ROUTINE Moldes   (* ladder *)
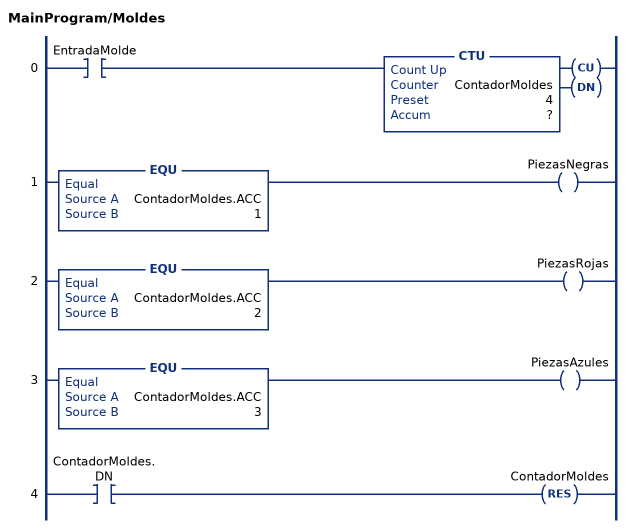
   0: XIC(EntradaMolde)CTU(ContadorMoldes,?,?);
   1: EQU(ContadorMoldes.ACC,1)OTE(PiezasNegras);
   2: EQU(ContadorMoldes.ACC,2)OTE(PiezasRojas);
   3: EQU(ContadorMoldes.ACC,3)OTE(PiezasAzules);
   4: XIC(ContadorMoldes.DN)RES(ContadorMoldes);
END_ROUTINE

ROUTINE ResetAll   (* sequential function chart *)
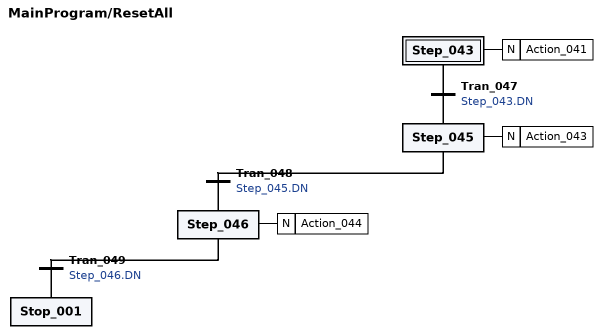
   INITIAL_STEP Step_043:
      ACTION Action_041 (N):
         Ruedas_Cero := 1;
         Chasis_Cero := 1;
         Inf_Cero := 1;
         Sup_Cero := 1;
         Ajuste_Cero := 1;
         Paredes_Cero := 1;
         Techo_Cero := 1;
         AjusteCasa_Cero := 1;
         Dispensar_Ruedas := 0;
         Dispensar_Chasis := 0;
         Dispensar_Inf := 0;
         Dispensar_Sup := 0;
         Dispensar_Timon := 0;
         Dispensar_Paredes := 0;
         Dispensar_Techo := 0;
         
      END_ACTION
   END_STEP
   TRANSITION Tran_047 FROM Step_043 TO Step_045
      := Step_043.DN
         
   END_TRANSITION
   STEP Step_045:
      ACTION Action_043 (N):
         TimerMoto_1.Reset := 1;
         TimerMoto_2.Reset := 1;
         TimerMoto_3.Reset := 1;
         TimerMoto_4.Reset := 1;
         TimerMoto_5.Reset := 1;
         TimerMoto_6.Reset := 1;
         TimerBarco_1.Reset := 1;
         TimerBarco_2.Reset := 1;
         TimerBarco_3.Reset := 1;
         TimerBarco_4.Reset := 1;
         TimerBarco_5.Reset := 1;
         TimerBarco_6.Reset := 1;
         TimerBarco_7.Reset := 1;
         TimerCasa_1.Reset := 1;
         TimerCasa_2.Reset := 1;
         TimerCasa_3.Reset := 1;
         TimerCasa_4.Reset := 1;
         TimerCasa_5.Reset := 1;
         TimerMoto_1.ACC := 0;
         TimerMoto_2.ACC := 0;
         TimerMoto_3.ACC := 0;
         TimerMoto_4.ACC := 0;
         TimerMoto_5.ACC := 0;
         TimerMoto_6.ACC := 0;
         TimerBarco_1.ACC := 0;
         TimerBarco_2.ACC := 0;
         TimerBarco_3.ACC := 0;
         TimerBarco_4.ACC := 0;
         TimerBarco_5.ACC := 0;
         TimerBarco_6.ACC := 0;
         TimerBarco_7.ACC := 0;
         TimerCasa_1.ACC := 0;
         TimerCasa_2.ACC := 0;
         TimerCasa_3.ACC := 0;
         TimerCasa_4.ACC := 0;
         TimerCasa_5.ACC := 0;
         TimerMoto_1.DN := 0;
         TimerMoto_2.DN := 0;
         TimerMoto_3.DN := 0;
         TimerMoto_4.DN := 0;
         TimerMoto_5.DN := 0;
         TimerMoto_6.DN := 0;
         TimerBarco_1.DN := 0;
         TimerBarco_2.DN := 0;
         TimerBarco_3.DN := 0;
         TimerBarco_4.DN := 0;
         TimerBarco_5.DN := 0;
         TimerBarco_6.DN := 0;
         TimerBarco_7.DN := 0;
         TimerCasa_1.DN := 0;
         TimerCasa_2.DN := 0;
         TimerCasa_3.DN := 0;
         TimerCasa_4.DN := 0;
         TimerCasa_5.DN := 0;
         
         TimerMoto_1.TimerEnable := 0;
         TimerMoto_2.TimerEnable := 0;
         TimerMoto_3.TimerEnable := 0;
         TimerMoto_4.TimerEnable := 0;
         TimerMoto_5.TimerEnable := 0;
         TimerMoto_6.TimerEnable := 0;
         TimerBarco_1.TimerEnable := 0;
         TimerBarco_2.TimerEnable := 0;
         TimerBarco_3.TimerEnable := 0;
         TimerBarco_4.TimerEnable := 0;
         TimerBarco_5.TimerEnable := 0;
         TimerBarco_6.TimerEnable := 0;
         TimerBarco_7.TimerEnable := 0;
         TimerCasa_1.TimerEnable := 0;
         TimerCasa_2.TimerEnable := 0;
         TimerCasa_3.TimerEnable := 0;
         TimerCasa_4.TimerEnable := 0;
         TimerCasa_5.TimerEnable := 0;
      END_ACTION
   END_STEP
   TRANSITION Tran_048 FROM Step_045 TO Step_046
      := Step_045.DN
   END_TRANSITION
   STEP Step_046:
      ACTION Action_044 (N):
         Action_000.Status:=0;
         Action_001.Status:=0;
         Action_002.Status:=0;
         Action_003.Status:=0;
         Action_004.Status:=0;
         Action_005.Status:=0;
         Action_006.Status:=0;
         Action_007.Status:=0;
         Action_008.Status:=0;
         Action_009.Status:=0;
         Action_010.Status:=0;
         Action_011.Status:=0;
         Action_012.Status:=0;
         Action_013.Status:=0;
         Action_014.Status:=0;
         Action_015.Status:=0;
         Action_016.Status:=0;
         Action_017.Status:=0;
         Action_018.Status:=0;
         Action_019.Status:=0;
         Action_020.Status:=0;
         Action_021.Status:=0;
         Action_022.Status:=0;
         Action_023.Status:=0;
         Action_024.Status:=0;
         Action_025.Status:=0;
         Action_026.Status:=0;
         Action_027.Status:=0;
         Action_028.Status:=0;
         Action_029.Status:=0;
         Action_030.Status:=0;
         Action_031.Status:=0;
         Action_032.Status:=0;
         Action_033.Status:=0;
         Action_034.Status:=0;
         Action_035.Status:=0;
         Action_036.Status:=0;
         Action_037.Status:=0;
         Action_038.Status:=0;
         
      END_ACTION
   END_STEP
   TRANSITION Tran_049 FROM Step_046 TO Stop_001
      := Step_046.DN
   END_TRANSITION
   STOP Stop_001;
END_ROUTINE
END_PROGRAM
